Fanuc TP program (LS listing): pcmove.ls

/PROG  PCMOVE
/ATTR
OWNER		= MNEDITOR;
COMMENT		= "";
PROG_SIZE	= 208;
CREATE		= DATE 26-09-22  TIME 10:06:56;
MODIFIED	= DATE 26-10-01  TIME 05:40:18;
FILE_NAME	= ;
VERSION		= 0;
LINE_COUNT	= 5;
MEMORY_SIZE	= 692;
PROTECT		= READ_WRITE;
TCD:  STACK_SIZE	= 0,
      TASK_PRIORITY	= 50,
      TIME_SLICE	= 0,
      BUSY_LAMP_OFF	= 0,
      ABORT_REQUEST	= 0,
      PAUSE_REQUEST	= 0;
DEFAULT_GROUP	= 1,*,*,*,*;
CONTROL_CODE	= 00000000 00000000;
/APPL
/MN
   1:  LBL[1] ;
   2:  WAIT DI[9]=ON    ;
   3:J PR[10:PC1] R[30]% FINE    ;
   4:  WAIT DI[9]=OFF    ;
   5:  JMP LBL[1] ;
/POS
/END
